TYPE ST_PMPS_Attenuator :
STRUCT
		nReqAtt : UINT;
		nAttCur : UINT;
		xAttOK : UINT;
END_STRUCT
END_TYPE

(* stored: Version 1.1.0.1, ProductVersion 3.1.4022.18
   DUT ST_PMPS_Attenuator: Id {91a12f52-7679-4a97-9c50-d3975974c134} *)
